RoboDK station: project-1.rdk

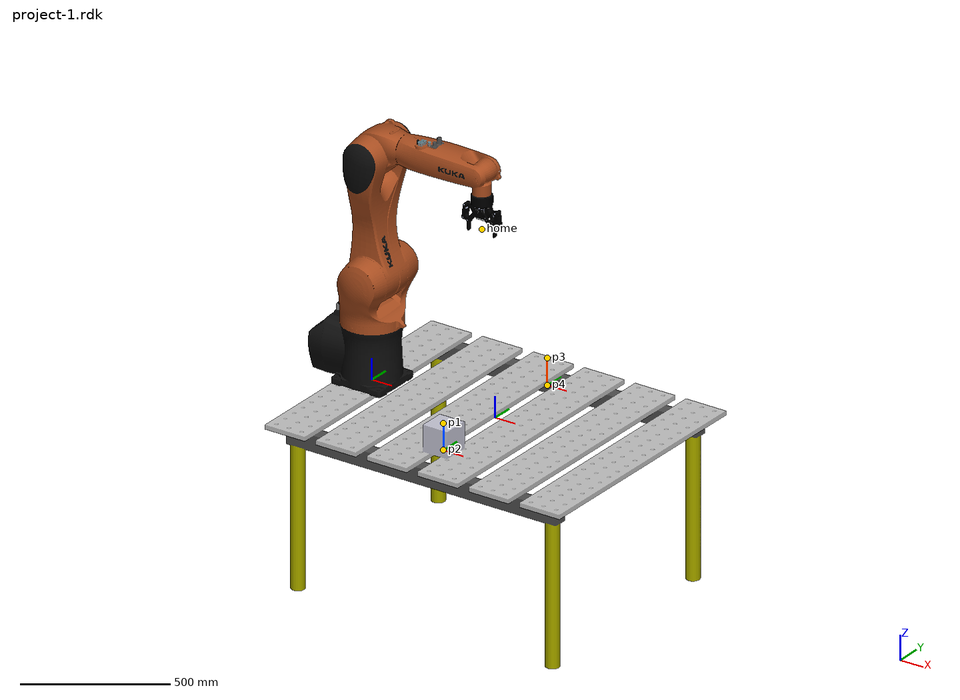
[picture v0: the station drawn from its stored meshes, robots at their saved joint values, targets as dots, program paths as lines]
Station project-1 (saved by RoboDK 5.8.0). Poses are relative to the parent item; angles as X-Y-Z fixed-axis rotations.
  - frame KUKA KR 10 R900 sixx Base at (-500, 0, 0) mm
    - robot KUKA KR 10 R900 sixx: 6 axes, payload 10 kg, reach 901 mm, repeatability 0.03 mm, weight 52 kg
        modified DH rows (alpha deg, a mm, theta deg, d mm): 0, 0, 0, 400; -90, 25, 0, 0; 0, 455, -90, 0; -90, 35, 0, 420; 90, 0, 0, 0; -90, 0, 180, 80
        joint limits [-170, -190, -120, -185, -120, -350] to [170, 45, 156, 185, 120, 350]; home [0, -90, 90, 0, 0, 0]; saved at [0, -90, 90, 0, 90, 0]
      - tool RobotiQ 2F-85 Gripper (Open), TCP at (0, 0, 130) mm, size 147.4 x 75 x 146.8 mm
  - frame base at (0, 0, 0) mm
    - object Table 1200x1000mm (Welding) at (0, 0, 0) mm, size 1193.8 x 965.2 x 609.6 mm, geometry from Table-1200x1000mm-Welding.sld
    - target home (Cartesian target) at (-55, 0, 680) mm, rotated rx 180 ry 0 rz -180 deg; joints [0, -90, 90, 0, 90, 0] of KUKA KR 10 R900 sixx
  - frame pick posittion at (0, -300, 0) mm
    - target p2 (Cartesian target) at (0, 0, 0) mm, rotated rx 180 ry 0 rz -180 deg; joints [30.964, -32.411, 102.794, 0, 19.616, 30.964] of KUKA KR 10 R900 sixx
    - target p1 (Cartesian target) at (0, 0, 100) mm, rotated rx 180 ry 0 rz -180 deg; joints [30.964, -43.632, 105.52, 0, 28.112, 30.964] of KUKA KR 10 R900 sixx
    - object box at (0, 0, 50) mm, size 100 x 100 x 100 mm, geometry from box.sld
  - frame place position at (0, 300, 0) mm
    - target p3 (Cartesian target) at (0, 0, 100) mm, rotated rx 180 ry 0 rz 180 deg; joints [-30.964, -43.632, 105.52, 0, 28.112, -30.964] of KUKA KR 10 R900 sixx
    - target p4 (Cartesian target) at (0, 0, 0) mm, rotated rx 180 ry 0 rz 180 deg; joints [-30.964, -32.411, 102.794, 0, 19.616, -30.964] of KUKA KR 10 R900 sixx
  - program restore (1 instructions, listed below)
  - program pick position (6 instructions, listed below)
  - program placing (6 instructions, listed below)
  - program main (8 instructions, listed below)
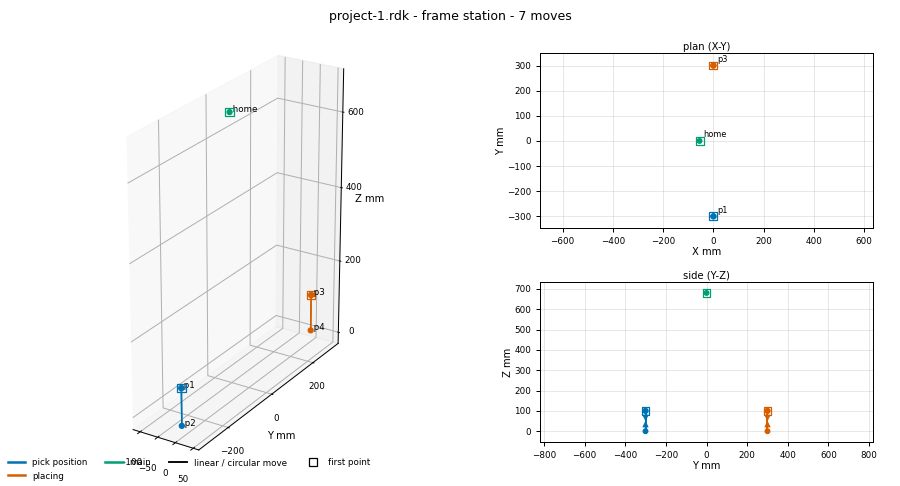
[picture p0: tool path of project-1.rdk in frame station, 7 of 7 moves have a stored position in this frame; points joined in program order, loops and branches not executed]

--- program restore (robot KUKA KR 10 R900 sixx) ---
  Replace objects

--- program pick position (robot KUKA KR 10 R900 sixx) ---
  Set Ref.: pick posittion
  Set Tool: RobotiQ 2F-85 Gripper (Open)
  MoveJ (p1)
  MoveL (p2)
  Attach to RobotiQ 2F-85 Gripper (Open)
  MoveL (p1)

--- program placing (robot KUKA KR 10 R900 sixx) ---
  Set Ref.: place position
  Set Tool: RobotiQ 2F-85 Gripper (Open)
  MoveJ (p3)
  MoveL (p4)
  Detach from RobotiQ 2F-85 Gripper (Open)
  MoveL (p3)

--- program main (robot KUKA KR 10 R900 sixx) ---
  Set Ref.: base
  Set Tool: RobotiQ 2F-85 Gripper (Open)
  MoveJ (home)
  Call restore
  Call pick position
  Call placing
  Set Ref.: base
  Call restore
